{attribute addProperty BoxType "EL1512-0000-0017"}
{attribute addProperty Id "CNT_Inputs_ChannelAT %I*ARRAY[0..1] OF CNT_Inputs_Channel_D5E647EE96120CNT_Outputs_ChannelAT %Q*ARRAY[0..1] OF CNT_Outputs_Channel_C7399CE196120WcStateAT %I*WcState_98A4DF7520.250InfoDataAT %I*InfoData_BC63D37F80100"}
{attribute addProperty CRC "2742845429"}
{attribute addProperty SizeInBites "274"}
{attribute addProperty SizeInBytes "34.25"}
TYPE EL1512_7D86CA5B :
STRUCT
	{attribute addProperty Name "CNT_Inputs_Channel"}
	CNT_Inputs_Channel : ARRAY[0..1] OF CNT_Inputs_Channel_D5E647EE;
	{attribute addProperty Name "CNT_Outputs_Channel"}
	CNT_Outputs_Channel : ARRAY[0..1] OF CNT_Outputs_Channel_C7399CE1;
	{attribute addProperty Name "WcState"}
	WcState : WcState_98A4DF75;
	{attribute addProperty Name "InfoData"}
	InfoData : InfoData_BC63D37F;
END_STRUCT
END_TYPE

(* stored: Version 1.2.0.0, ProductVersion 3.1.4024.9
   DUT EL1512_7D86CA5B: Id {af365e3a-60d5-486b-a5ec-d9dc79f4fe51} *)
